(* CoDeSys 2.3.5.6 project: calaos_ethernet.pro *)
(* Libraries: Ethernet.lib*2.12.10 13:48:36, Standard.lib 2.12.10 13:48:36 *)

(* PLC configuration (modules and I/O channels)
0750-0530 8 DO 24 V DC 0.5A [Type_10_8_Channels] node 0, in %IB0 out %QB0
  AT %QX0.0 [BOOLOnX_Q] Ch_1 Digital output
  AT %QX0.1 [BOOLOnX_Q] Ch_2 Digital output
  AT %QX0.2 [BOOLOnX_Q] Ch_3 Digital output
  AT %QX0.3 [BOOLOnX_Q] Ch_4 Digital output
  AT %QX0.4 [BOOLOnX_Q] Ch_5 Digital output
  AT %QX0.5 [BOOLOnX_Q] Ch_6 Digital output
  AT %QX0.6 [BOOLOnX_Q] Ch_7 Digital output
  AT %QX0.7 [BOOLOnX_Q] Ch_8 Digital output
0750-0530 8 DO 24 V DC 0.5A [Type_10_8_Channels] node 0, in %IB0 out %QB0
  AT %QX0.8 [BOOLOnX_Q] Ch_1 Digital output
  AT %QX0.9 [BOOLOnX_Q] Ch_2 Digital output
  AT %QX0.10 [BOOLOnX_Q] Ch_3 Digital output
  AT %QX0.11 [BOOLOnX_Q] Ch_4 Digital output
  AT %QX0.12 [BOOLOnX_Q] Ch_5 Digital output
  AT %QX0.13 [BOOLOnX_Q] Ch_6 Digital output
  AT %QX0.14 [BOOLOnX_Q] Ch_7 Digital output
  AT %QX0.15 [BOOLOnX_Q] Ch_8 Digital output
0750-0530 8 DO 24 V DC 0.5A [Type_10_8_Channels] node 0, in %IB0 out %QB0
  AT %QX1.0 [BOOLOnX_Q] Ch_1 Digital output
  AT %QX1.1 [BOOLOnX_Q] Ch_2 Digital output
  AT %QX1.2 [BOOLOnX_Q] Ch_3 Digital output
  AT %QX1.3 [BOOLOnX_Q] Ch_4 Digital output
  AT %QX1.4 [BOOLOnX_Q] Ch_5 Digital output
  AT %QX1.5 [BOOLOnX_Q] Ch_6 Digital output
  AT %QX1.6 [BOOLOnX_Q] Ch_7 Digital output
  AT %QX1.7 [BOOLOnX_Q] Ch_8 Digital output
0750-0530 8 DO 24 V DC 0.5A [Type_10_8_Channels] node 0, in %IB0 out %QB0
  AT %QX1.8 [BOOLOnX_Q] Ch_1 Digital output
  AT %QX1.9 [BOOLOnX_Q] Ch_2 Digital output
  AT %QX1.10 [BOOLOnX_Q] Ch_3 Digital output
  AT %QX1.11 [BOOLOnX_Q] Ch_4 Digital output
  AT %QX1.12 [BOOLOnX_Q] Ch_5 Digital output
  AT %QX1.13 [BOOLOnX_Q] Ch_6 Digital output
  AT %QX1.14 [BOOLOnX_Q] Ch_7 Digital output
  AT %QX1.15 [BOOLOnX_Q] Ch_8 Digital output
0750-0530 8 DO 24 V DC 0.5A [Type_10_8_Channels] node 0, in %IB0 out %QB0
  AT %QX2.0 [BOOLOnX_Q] Ch_1 Digital output
  AT %QX2.1 [BOOLOnX_Q] Ch_2 Digital output
  AT %QX2.2 [BOOLOnX_Q] Ch_3 Digital output
  AT %QX2.3 [BOOLOnX_Q] Ch_4 Digital output
  AT %QX2.4 [BOOLOnX_Q] Ch_5 Digital output
  AT %QX2.5 [BOOLOnX_Q] Ch_6 Digital output
  AT %QX2.6 [BOOLOnX_Q] Ch_7 Digital output
  AT %QX2.7 [BOOLOnX_Q] Ch_8 Digital output
0750-0530 8 DO 24 V DC 0.5A [Type_10_8_Channels] node 0, in %IB0 out %QB0
  AT %QX2.8 [BOOLOnX_Q] Ch_1 Digital output
  AT %QX2.9 [BOOLOnX_Q] Ch_2 Digital output
  AT %QX2.10 [BOOLOnX_Q] Ch_3 Digital output
  AT %QX2.11 [BOOLOnX_Q] Ch_4 Digital output
  AT %QX2.12 [BOOLOnX_Q] Ch_5 Digital output
  AT %QX2.13 [BOOLOnX_Q] Ch_6 Digital output
  AT %QX2.14 [BOOLOnX_Q] Ch_7 Digital output
  AT %QX2.15 [BOOLOnX_Q] Ch_8 Digital output
0750-0530 8 DO 24 V DC 0.5A [Type_10_8_Channels] node 0, in %IB0 out %QB0
  AT %QX3.0 [BOOLOnX_Q] Ch_1 Digital output
  AT %QX3.1 [BOOLOnX_Q] Ch_2 Digital output
  AT %QX3.2 [BOOLOnX_Q] Ch_3 Digital output
  AT %QX3.3 [BOOLOnX_Q] Ch_4 Digital output
  AT %QX3.4 [BOOLOnX_Q] Ch_5 Digital output
  AT %QX3.5 [BOOLOnX_Q] Ch_6 Digital output
  AT %QX3.6 [BOOLOnX_Q] Ch_7 Digital output
  AT %QX3.7 [BOOLOnX_Q] Ch_8 Digital output
0750-0530 8 DO 24 V DC 0.5A [Type_10_8_Channels] node 0, in %IB0 out %QB0
  AT %QX3.8 [BOOLOnX_Q] Ch_1 Digital output
  AT %QX3.9 [BOOLOnX_Q] Ch_2 Digital output
  AT %QX3.10 [BOOLOnX_Q] Ch_3 Digital output
  AT %QX3.11 [BOOLOnX_Q] Ch_4 Digital output
  AT %QX3.12 [BOOLOnX_Q] Ch_5 Digital output
  AT %QX3.13 [BOOLOnX_Q] Ch_6 Digital output
  AT %QX3.14 [BOOLOnX_Q] Ch_7 Digital output
  AT %QX3.15 [BOOLOnX_Q] Ch_8 Digital output
0750-0530 8 DO 24 V DC 0.5A [Type_10_8_Channels] node 0, in %IB0 out %QB0
  AT %QX4.0 [BOOLOnX_Q] Ch_1 Digital output
  AT %QX4.1 [BOOLOnX_Q] Ch_2 Digital output
  AT %QX4.2 [BOOLOnX_Q] Ch_3 Digital output
  AT %QX4.3 [BOOLOnX_Q] Ch_4 Digital output
  AT %QX4.4 [BOOLOnX_Q] Ch_5 Digital output
  AT %QX4.5 [BOOLOnX_Q] Ch_6 Digital output
  AT %QX4.6 [BOOLOnX_Q] Ch_7 Digital output
  AT %QX4.7 [BOOLOnX_Q] Ch_8 Digital output
0750-0530 8 DO 24 V DC 0.5A [Type_10_8_Channels] node 0, in %IB0 out %QB0
  AT %QX4.8 [BOOLOnX_Q] Ch_1 Digital output
  AT %QX4.9 [BOOLOnX_Q] Ch_2 Digital output
  AT %QX4.10 [BOOLOnX_Q] Ch_3 Digital output
  AT %QX4.11 [BOOLOnX_Q] Ch_4 Digital output
  AT %QX4.12 [BOOLOnX_Q] Ch_5 Digital output
  AT %QX4.13 [BOOLOnX_Q] Ch_6 Digital output
  AT %QX4.14 [BOOLOnX_Q] Ch_7 Digital output
  AT %QX4.15 [BOOLOnX_Q] Ch_8 Digital output
0750-0430 8 DI 24 V DC 3.0ms [Type_1_8_Channels] node 0, in %IB0 out %QB0
  AT %IX4.0 [BOOLOnX_I] Ch_1 Digital input
  AT %IX4.1 [BOOLOnX_I] Ch_2 Digital input
  AT %IX4.2 [BOOLOnX_I] Ch_3 Digital input
  AT %IX4.3 [BOOLOnX_I] Ch_4 Digital input
  AT %IX4.4 [BOOLOnX_I] Ch_5 Digital input
  AT %IX4.5 [BOOLOnX_I] Ch_6 Digital input
  AT %IX4.6 [BOOLOnX_I] Ch_7 Digital input
  AT %IX4.7 [BOOLOnX_I] Ch_8 Digital input
0750-0430 8 DI 24 V DC 3.0ms [Type_1_8_Channels] node 0, in %IB0 out %QB0
  AT %IX4.8 [BOOLOnX_I] Ch_1 Digital input
  AT %IX4.9 [BOOLOnX_I] Ch_2 Digital input
  AT %IX4.10 [BOOLOnX_I] Ch_3 Digital input
  AT %IX4.11 [BOOLOnX_I] Ch_4 Digital input
  AT %IX4.12 [BOOLOnX_I] Ch_5 Digital input
  AT %IX4.13 [BOOLOnX_I] Ch_6 Digital input
  AT %IX4.14 [BOOLOnX_I] Ch_7 Digital input
  AT %IX4.15 [BOOLOnX_I] Ch_8 Digital input
0750-0430 8 DI 24 V DC 3.0ms [Type_1_8_Channels] node 0, in %IB0 out %QB0
  AT %IX5.0 [BOOLOnX_I] Ch_1 Digital input
  AT %IX5.1 [BOOLOnX_I] Ch_2 Digital input
  AT %IX5.2 [BOOLOnX_I] Ch_3 Digital input
  AT %IX5.3 [BOOLOnX_I] Ch_4 Digital input
  AT %IX5.4 [BOOLOnX_I] Ch_5 Digital input
  AT %IX5.5 [BOOLOnX_I] Ch_6 Digital input
  AT %IX5.6 [BOOLOnX_I] Ch_7 Digital input
  AT %IX5.7 [BOOLOnX_I] Ch_8 Digital input
0750-0430 8 DI 24 V DC 3.0ms [Type_1_8_Channels] node 0, in %IB0 out %QB0
  AT %IX5.8 [BOOLOnX_I] Ch_1 Digital input
  AT %IX5.9 [BOOLOnX_I] Ch_2 Digital input
  AT %IX5.10 [BOOLOnX_I] Ch_3 Digital input
  AT %IX5.11 [BOOLOnX_I] Ch_4 Digital input
  AT %IX5.12 [BOOLOnX_I] Ch_5 Digital input
  AT %IX5.13 [BOOLOnX_I] Ch_6 Digital input
  AT %IX5.14 [BOOLOnX_I] Ch_7 Digital input
  AT %IX5.15 [BOOLOnX_I] Ch_8 Digital input
0750-0430 8 DI 24 V DC 3.0ms [Type_1_8_Channels] node 0, in %IB0 out %QB0
  AT %IX6.0 [BOOLOnX_I] Ch_1 Digital input
  AT %IX6.1 [BOOLOnX_I] Ch_2 Digital input
  AT %IX6.2 [BOOLOnX_I] Ch_3 Digital input
  AT %IX6.3 [BOOLOnX_I] Ch_4 Digital input
  AT %IX6.4 [BOOLOnX_I] Ch_5 Digital input
  AT %IX6.5 [BOOLOnX_I] Ch_6 Digital input
  AT %IX6.6 [BOOLOnX_I] Ch_7 Digital input
  AT %IX6.7 [BOOLOnX_I] Ch_8 Digital input
0750-0430 8 DI 24 V DC 3.0ms [Type_1_8_Channels] node 0, in %IB0 out %QB0
  AT %IX6.8 [BOOLOnX_I] Ch_1 Digital input
  AT %IX6.9 [BOOLOnX_I] Ch_2 Digital input
  AT %IX6.10 [BOOLOnX_I] Ch_3 Digital input
  AT %IX6.11 [BOOLOnX_I] Ch_4 Digital input
  AT %IX6.12 [BOOLOnX_I] Ch_5 Digital input
  AT %IX6.13 [BOOLOnX_I] Ch_6 Digital input
  AT %IX6.14 [BOOLOnX_I] Ch_7 Digital input
  AT %IX6.15 [BOOLOnX_I] Ch_8 Digital input
0750-1405 16 DI 24V DC 3.0ms [Type_1_16_Channels] node 0, in %IB0 out %QB0
  AT %IX7.0 [BOOLOnX_I] Ch_1 Digital input
  AT %IX7.1 [BOOLOnX_I] Ch_2 Digital input
  AT %IX7.2 [BOOLOnX_I] Ch_3 Digital input
  AT %IX7.3 [BOOLOnX_I] Ch_4 Digital input
  AT %IX7.4 [BOOLOnX_I] Ch_5 Digital input
  AT %IX7.5 [BOOLOnX_I] Ch_6 Digital input
  AT %IX7.6 [BOOLOnX_I] Ch_7 Digital input
  AT %IX7.7 [BOOLOnX_I] Ch_8 Digital input
  AT %IX7.8 [BOOLOnX_I] Ch_9 Digital input
  AT %IX7.9 [BOOLOnX_I] Ch_10 Digital input
  AT %IX7.10 [BOOLOnX_I] Ch_11 Digital input
  AT %IX7.11 [BOOLOnX_I] Ch_12 Digital input
  AT %IX7.12 [BOOLOnX_I] Ch_13 Digital input
  AT %IX7.13 [BOOLOnX_I] Ch_14 Digital input
  AT %IX7.14 [BOOLOnX_I] Ch_15 Digital input
  AT %IX7.15 [BOOLOnX_I] Ch_16 Digital input
0750-0460/0000-0003 4 AI PT1000 (RTD) [Type_44_4_Channels] node 0, in %IB0 out %QB0
  AT %IW0 [INTOnW_I] Ch_1 signed Input value
  AT %IW1 [INTOnW_I] Ch_2 signed Input value
  AT %IW2 [INTOnW_I] Ch_3 signed Input value
  AT %IW3 [INTOnW_I] Ch_4 signed Input value
Fieldbus variables [FB_VARS] node 1, in %IB0 out %QB0
Flag variables [FLAG_VARS] node 2, in %IB0 out %QB0
*)

(* Data type *)
TYPE typEthernet_BUFFER :
	STRUCT
		Index		:	INT;
		Data		:	ARRAY[1..1500] OF BYTE;
	END_STRUCT
END_TYPE

(* POU PLC_PRG, ST *)
PROGRAM PLC_PRG
VAR
	(* Calaos Client *)
	CalaosClient: Calaos_Ethernet_Client;
	ReceiveData: typEthernet_buffer;
	StartSendClient: BOOL := FALSE;

	(* Calaos Input Status *)
	CalaosInput: Calaos_Ethernet_Input;
	StartSendInput: BOOL := FALSE;
	InputNum: BYTE;
	InputStatus: BOOL;

	(* Config *)
	ServerIP: STRING := '10.0.0.200';
	CalaosUsername: STRING := 'username';
	CalaosPassword: STRING := 'pass';

	Command: STRING(255);

	InputAddr1 AT %IX6.0: BOOL;
	Input1: INTER_EVENT;

	InputAddr2 AT %IX6.2: BOOL;
	Input2: INTER_EVENT;

END_VAR
Input1(IN := InputAddr1);
Input2(IN := InputAddr2);

(* Read inputs and send their status on the network if they changed *)
IF (Input1.ON = TRUE) THEN
	(* Send command to calaos server if Input2 is pressed *)
	Command := 'output input_1 set true';
	StartSendClient := TRUE;
END_IF


IF (Input2.ON = TRUE) THEN
	(* Send input state change to Calaos *)
	InputNum := 2;
	InputStatus := TRUE; (* input status changed to true *)
	StartSendInput := TRUE;
END_IF
IF (Input2.OFF = TRUE) THEN
	(* Send input state change to Calaos *)
	InputNum := 2;
	InputStatus := FALSE; (* input status changed to false *)
	StartSendInput := TRUE;
END_IF


(* send command to calaos server *)
CalaosClient(xOpen := TRUE,
		wIP := IP_ADDRESS(ServerIP),
		Login := CalaosUsername,
		Pass := CalaosPassword,
		Command := Command,
		ReceiveBuff := ReceiveData,
		xStartSend := StartSendClient);

(* send input status to calaos server *)
CalaosInput(xOpen := TRUE,
		wIP := IP_ADDRESS(ServerIP),
		Input := InputNum,
		InputState := InputStatus,
		xStartSend := StartSendInput);
END_PROGRAM

(* POU Calaos_Ethernet_Client, ST *)
FUNCTION_BLOCK Calaos_Ethernet_Client
(*
	Calaos_Ethernet_Client
	Envoi de commande à un serveur Calaos, avec gestion de l'authentification
	Les commandes sont les meme que spécifié ici: http://support.calaos.fr/protocole_tcp
*)
VAR_INPUT
	xOpen: BOOL;						(* TRUE active le client *)
	wIP: DWORD;							(* Adresse IP du serveur Calaos *)
	Login: STRING(255);					(* Username pour l'authentification *)
	Pass: STRING(255);					(* Mot de passe pour l'authentification *)
	Command: STRING(255);				(* Commande à envoyer. Ex: "output output_23 set true" *)
END_VAR
VAR_IN_OUT
	xStartSend: BOOL;					(* Mettre à true pour commencer la transmission, remis à FALSE quand la transmission est terminé *)
	ReceiveBuff: typEthernet_BUFFER;	(* Receive Buffer *)
END_VAR
VAR_OUTPUT
	Error: ETH_ERROR;					(* <> NO_ERROR si erreur *)
	xConnected:	BOOL;					(* TRUE si la connection est établie *)
	xDataReceived: BOOL;				(* front montant si des données ont été recus *)
	Socket: WORD;						(* Socket de communication *)
END_VAR
VAR
	SocketOpen: ETHERNET_CLIENT_OPEN;
	SocketClose: ETHERNET_CLIENT_CLOSE;
	SocketWrite: ETHERNET_WRITE_PT;
	SocketRead: ETHERNET_READ;
	EthernetBuffer: ARRAY[1..1500] OF BYTE;
	Status: WORD:=0;
	i: INT;
	GetNetConfig: ETHERNET_GET_NETWORK_CONFIG;
	CloseStatus: INT;
	cmd: STRING(255);
	pBuffer: POINTER TO BYTE;
END_VAR
IF xOpen THEN

	CASE Status OF
		0: (* Init *)
			GetNetConfig(EN := FALSE);
			GetNetConfig(EN := TRUE);
			Status := 4;
			Error := NO_ERROR;
			Socket := 0;
			CloseStatus:=0;
			xConnected := FALSE;
			xDataReceived := FALSE;

		1: (* Wait for init *)
			GetNetConfig(EN := TRUE);
			IF GetNetConfig.ENO THEN
				IF GetNetConfig.IP_ADR <> 0 THEN
					Status := 4; (* Init done *)
				ELSE
					Status := 0; (* try again *)
				END_IF
			END_IF

		4: (* Open connection *)
			SocketRead(EN := 0, SOCKET := 0, DATA := EthernetBuffer);
			SocketClose(EN := 0);
			SocketOpen(EN := 0);

			SocketOpen(EN := 1, TYP := SOCK_STREAM, PROTO:= IPPROTO_TCP, IP_ADR:= wIP, PORT := 4456);

			Status := 5;

		5: (* Wait for connection *)
			SocketOpen(EN := 1, TYP := SOCK_STREAM, PROTO:= IPPROTO_TCP, IP_ADR:= wIP, PORT := 4456);

			IF SocketOpen.ENO = 1 THEN
				IF SocketOpen.ERROR = NO_ERROR THEN
					Status := 6; (* Connection successfull *)
					xConnected := TRUE;
					Socket := SocketOpen.SOCKET;

					(* Set up the login command *)
					cmd := 'login ';
					cmd := CONCAT(cmd, Login);
					cmd := CONCAT(cmd, ' ');
					cmd := CONCAT(cmd, Pass);
					cmd := CONCAT(cmd, '$R$n');
				ELSE
					Status := 0; (* Error, try again *)
				END_IF;
				Error := SocketOpen.ERROR;
			END_IF

		6: (* Send login command to authenticate *)
			pBuffer := ADR(cmd);
			SocketWrite(EN := 1,
						SOCKET := Socket,
						LEN_IN := LEN(cmd) + 1,
						DATA_PT := pBuffer);

			IF SocketWrite.ENO THEN
				IF(SocketWrite.ERROR <> NO_ERROR) THEN
					Status := 40; (* Error writing to the socket, close it *)
				ELSE
					Status := 10; (* Login complete, wait to read data *)
				END_IF;
				Error := SocketWrite.ERROR;
			END_IF

		10: (* Wait for data to read *)

	 		SocketRead(EN := 1, SOCKET := Socket, DATA := EthernetBuffer);
			SocketRead(EN := 0, SOCKET := 0, DATA := EthernetBuffer);

			Error := SocketRead.ERROR;
			IF(SocketRead.ERROR <> NO_ERROR) THEN (* Error reading the socket, close it *)
				Status := 40;
			ELSIF (SocketRead.LEN_OUT <> 0) THEN (* Read some new data *)
				Status := 20;
				xDataReceived := FALSE;
			ELSIF (LEN(Command) > 0 AND xStartSend) THEN (* We have data to send *)
				Status := 30;
				SocketWrite(EN := 0, DATA_PT := pBuffer);

				(* prepare command *)
				cmd := '';
				cmd := CONCAT(cmd, Command);
				cmd := CONCAT(cmd, '$R$n');
			END_IF

		20:	(* Copy the data received to the receive buffer *)

			FOR i := 1 TO SocketRead.LEN_OUT DO
				ReceiveBuff.index := (ReceiveBuff.index MOD 1500) + 1;
				ReceiveBuff.data[ReceiveBuff.index] := EthernetBuffer[i];
			END_FOR
			Status := 10;
			xDataReceived := TRUE;

		30: (* Send data to peer *)

			pBuffer := ADR(cmd);
			SocketWrite(EN := 1,
						SOCKET := Socket,
						LEN_IN := LEN(cmd) + 1,
						DATA_PT := pBuffer);

			IF SocketWrite.ENO THEN
				IF(SocketWrite.ERROR <> NO_ERROR) THEN
					Status := 40; (* Error writing to the socket, close it *)
				ELSE
					Status := 10; (* Login complete, wait to read data *)
				END_IF;
				Error := SocketWrite.ERROR;
				xStartSend := FALSE;
			END_IF

		40:	(* Close the socket *)

			SocketClose(EN := 1, SOCKET := Socket);
			IF SocketClose.ENO THEN
				SocketClose(EN := 0);
				xConnected := FALSE;
				Status := 0; (* Restart from the begining *)
			END_IF
	
	END_CASE;
ELSE
	CASE CloseStatus OF
	0:
		SocketClose(EN := 0);
		SocketClose(EN := 1, SOCKET:= Socket);
		CloseStatus := 1;
	1:
		SocketClose(EN := 1, SOCKET:= Socket);
		IF SocketClose.ENO THEN
			SocketClose(EN := 0);
			CloseStatus := 2;
		END_IF
	2:
		Status := 0;
		Error := NO_ERROR;
		xConnected := FALSE;
		xDataReceived := FALSE;
	END_CASE
END_IF
END_FUNCTION_BLOCK

(* POU Calaos_Ethernet_Input, ST *)
FUNCTION_BLOCK Calaos_Ethernet_Input
(*
	Calaos_Ethernet_Input
	Envoi le changement d'etat d'une entrée à un serveur Calaos
*)
VAR_INPUT
	xOpen: BOOL;						(* TRUE active le client *)
	wIP: DWORD;							(* Adresse IP du serveur Calaos *)
	Input: BYTE;						(* numéro de l'entrée à envoyer *)
	InputState: BOOL;					(* Etat de l'entrée *)
END_VAR
VAR_IN_OUT
	xStartSend: BOOL;					(* Mettre à true pour commencer la transmission, remis à FALSE quand la transmission est terminé *)
END_VAR
VAR_OUTPUT
	Error: ETH_ERROR;					(* <> NO_ERROR si erreur *)
	Socket: WORD;						(* Socket de communication *)
END_VAR
VAR
	SocketOpen: ETHERNET_CLIENT_OPEN;
	SocketClose: ETHERNET_CLIENT_CLOSE;
	SocketWrite: ETHERNET_WRITE_PT;
	SocketRead: ETHERNET_READ;
	EthernetBuffer: ARRAY[1..1500] OF BYTE;
	Status: WORD:=0;
	i: INT;
	GetNetConfig: ETHERNET_GET_NETWORK_CONFIG;
	CloseStatus: INT;
	cmd: STRING(255);
	pBuffer: POINTER TO BYTE;
	ReceiveBuff: typEthernet_BUFFER;	(* Receive Buffer *)
END_VAR
IF xOpen THEN

	CASE Status OF
		0: (* Init *)
			GetNetConfig(EN := FALSE);
			GetNetConfig(EN := TRUE);
			Status := 4;
			Error := NO_ERROR;
			Socket := 0;
			CloseStatus:=0;

		1: (* Wait for init *)
			GetNetConfig(EN := TRUE);
			IF GetNetConfig.ENO THEN
				IF GetNetConfig.IP_ADR <> 0 THEN
					Status := 4; (* Init done *)
				ELSE
					Status := 0; (* try again *)
				END_IF
			END_IF

		4: (* Open connection *)
			SocketRead(EN := 0, SOCKET := 0, DATA := EthernetBuffer);
			SocketClose(EN := 0);
			SocketOpen(EN := 0);

			SocketOpen(EN := 1, TYP := SOCK_DGRAM, PROTO:= IPPROTO_UDP, IP_ADR:= wIP, PORT := 4646);

			Status := 5;

		5: (* Wait for connection *)
			SocketOpen(EN := 1, TYP := SOCK_STREAM, PROTO:= IPPROTO_TCP, IP_ADR:= wIP, PORT := 4646);

			IF SocketOpen.ENO = 1 THEN
				IF SocketOpen.ERROR = NO_ERROR THEN
					Status := 10; (* Connection successfull *)
					Socket := SocketOpen.SOCKET;
				ELSE
					Status := 0; (* Error, try again *)
				END_IF;
				Error := SocketOpen.ERROR;
			END_IF

		10: (* Wait for data to read (don't use these data, just read them to empty the Ethernet Buffer) *)

	 		SocketRead(EN := 1, SOCKET := Socket, DATA := EthernetBuffer);
			SocketRead(EN := 0, SOCKET := 0, DATA := EthernetBuffer);

			Error := SocketRead.ERROR;
			IF(SocketRead.ERROR <> NO_ERROR) THEN (* Error reading the socket, close it *)
				Status := 40;
			ELSIF (SocketRead.LEN_OUT <> 0) THEN (* Read some new data *)
				Status := 20;
			ELSIF (xStartSend) THEN (* We have data to send *)
				Status := 30;
				SocketWrite(EN := 0, DATA_PT := pBuffer);

				(* prepare command *)
				cmd := 'WAGO INT ';
				cmd := CONCAT(cmd, BYTE_TO_STRING(Input));
				IF InputState = TRUE THEN
					cmd := CONCAT(cmd, ' 1');
				ELSE
					cmd := CONCAT(cmd, ' 0');
				END_IF
			END_IF

		20:	(* Don't do anything with the data read *)
			Status := 10;

		30: (* Send data to peer *)

			pBuffer := ADR(cmd);
			SocketWrite(EN := 1,
						SOCKET := Socket,
						LEN_IN := LEN(cmd) + 1,
						DATA_PT := pBuffer);

			IF SocketWrite.ENO THEN
				IF(SocketWrite.ERROR <> NO_ERROR) THEN
					Status := 40; (* Error writing to the socket, close it *)
				ELSE
					Status := 10; (* Login complete, wait to read data *)
				END_IF;
				Error := SocketWrite.ERROR;
				xStartSend := FALSE;
			END_IF

		40:	(* Close the socket *)

			SocketClose(EN := 1, SOCKET := Socket);
			IF SocketClose.ENO THEN
				SocketClose(EN := 0);
				Status := 0; (* Restart from the begining *)
			END_IF

	END_CASE;
ELSE
	CASE CloseStatus OF
	0:
		SocketClose(EN := 0);
		SocketClose(EN := 1, SOCKET:= Socket);
		CloseStatus := 1;
	1:
		SocketClose(EN := 1, SOCKET:= Socket);
		IF SocketClose.ENO THEN
			SocketClose(EN := 0);
			CloseStatus := 2;
		END_IF
	2:
		Status := 0;
		Error := NO_ERROR;
	END_CASE
END_IF
END_FUNCTION_BLOCK

(* POU INTER_EVENT, ST *)
FUNCTION_BLOCK INTER_EVENT
VAR_INPUT
	IN: BOOL;
END_VAR
VAR_OUTPUT
	ON: BOOL;
	OFF: BOOL;
END_VAR
VAR
	MTRIG: R_TRIG;
	DTRIG: F_TRIG;
END_VAR
(* Detection de front montant et descendant sur une entrée *)

MTRIG(CLK := IN);
ON := MTRIG.Q;
DTRIG(CLK := IN);
OFF := DTRIG.Q;
END_FUNCTION_BLOCK

(* POU IP_ADDRESS, ST *)
FUNCTION IP_ADDRESS : DWORD
VAR_INPUT
	IP_ADR	:	STRING;
END_VAR
VAR
	Address 	:	DWORD;
	Value		:	WORD;
	DecimalPos	:	INT;
	Rest		:	STRING;
END_VAR
Address := STRING_TO_WORD(IP_ADR);
IF (Address <= 255) AND (Address >= 0) THEN
	DecimalPos := FIND(IP_ADR,'.');
	IF DecimalPos <> 0 THEN
		Rest := RIGHT(IP_ADR,LEN(IP_ADR) - DecimalPos);
		Value := STRING_TO_WORD(Rest);
		IF (Value <= 255) AND (Value >= 0) THEN
			Address := (Address * 16#0100) + Value;

			DecimalPos := FIND(Rest,'.');
			IF DecimalPos <> 0 THEN
				Rest := RIGHT(IP_ADR,LEN(Rest) - DecimalPos);
				Value := STRING_TO_WORD(Rest);
				IF (Value <= 255) AND (Value >= 0) THEN
					Address := (Address * 16#0100) + Value;

					DecimalPos := FIND(Rest,'.');
					IF DecimalPos <> 0 THEN
						Rest := RIGHT(IP_ADR,LEN(Rest) - DecimalPos);
						Value := STRING_TO_WORD(Rest);
						IF (Value <= 255) AND (Value >= 0) THEN
							Address := (Address * 16#0100) + Value;
						ELSE
							Address := 0;
						END_IF
					ELSE
						Address := 0;
					END_IF
				ELSE
					Address := 0;
				END_IF
			ELSE
				Address := 0;
			END_IF
		ELSE
			Address := 0;
		END_IF
	ELSE
		Address := 0;
	END_IF
ELSE
	Address := 0;
END_IF
IP_Address := Address;
END_FUNCTION
